(* IEC 61131-3 sources: Industry-PLC-LLM/data/PLCBEAD_repo/PLCBEAD_PLCEmbed-main/PLC-BEAD/Source/GEB/AGDF, 1 file *)

(* ---- AGDF.ST ---- *)
FUNCTION AGDF:REAL
	VAR_INPUT
		X :	REAL;
	END_VAR

	AGDF := LN((1.0 + SIN(X)) / COS(X));
END_FUNCTION

PROGRAM program0
  VAR
    LocalVar0 : REAL;
    LocalOUT  : REAL;
  END_VAR

  LocalOUT := AGDF(LocalVar0);
END_PROGRAM
